{attribute 'hide'}
FUNCTION F_HwSetAddrInfo_29bit_CX2500_M510 : ST_CanData_29bit_CX2500_M510
VAR_INPUT
	stInput: ST_CanHeader;
END_VAR

F_HwSetAddrInfo_29bit_CX2500_M510.nCobid := 16#3FFFFFFF AND stInput.nCobid;

IF (stInput.nCobid > 16#7FF AND NOT stInput.bExtendedAddress) THEN // check cobid and extended address flags is set correctly
	stInput.bExtendedAddress := TRUE;//fix issue
END_IF

F_HwSetAddrInfo_29bit_CX2500_M510.nCobid.31 := stInput.bExtendedAddress;//sets extended address flag, if set raw can message will have 29bit for identification on the wire.

F_HwSetAddrInfo_29bit_CX2500_M510.nCobid.30 := stInput.bRTR;// sets RTR bit

IF (stInput.nMsgLength > 8) THEN
	F_HwSetAddrInfo_29bit_CX2500_M510.nLength := 8;
ELSE
	F_HwSetAddrInfo_29bit_CX2500_M510.nLength := stInput.nMsgLength;
END_IF

END_FUNCTION

(* stored: Version 1.1.0.1, ProductVersion 3.1.4024.12
   POU F_HwSetAddrInfo_29bit_CX2500_M510: Id {dbfe778d-d3d6-01fc-1261-9217a36ba26b}, SpecialFunc None *)
